# EPICS substitutions: iocs/simple-power-pmac/labApp/Db/lab_expanded.substitutions
# This file was automatically generated on Fri 25 May 2018 08:06:14 BST from
# source: /home/hgv27681/R3.14.12.3/support/pmac/etc/makeIocs/lab.xml
#
# *** Please do not edit this file: edit the source file instead. ***
#

# Macros:
#  PORT      The asyn port for the pmac controller
#  P         PV Prefix
#  NAXES     Number of axes
#  TIMEOUT   Timeout for controller communication
#  FEEDRATE  feedrate below which we go into error
#  CSG0      Name for Coordinate System Group 0
#  CSG1      Name for Coordinate System Group 1
#  CSG2      Name for Coordinate System Group 2
#  CSG3      Name for Coordinate System Group 3
#  CSG4      Name for Coordinate System Group 4
#  CSG5      Name for Coordinate System Group 5
#  CSG6      Name for Coordinate System Group 6
#  CSG7      Name for Coordinate System Group 7
file $(PMAC)/db/pmacController.template
{
pattern { PORT, P, NAXES, TIMEOUT, FEEDRATE, CSG0, CSG1, CSG2, CSG3, CSG4, CSG5, CSG6, CSG7 }
    { "Brick", "BRICK1", "8", "4", "100", "", "", "", "", "", "", "", "" }
}

# Macros:
#  PORT  The asyn port for the pmac controller
#  P     PV Prefix
file $(PMAC)/db/powerPmacStatus.template
{
pattern { PORT, P }
    { "Brick", "BRICK1" }
}

# Macros:
#  PMAC  Pmac/Geobrick name
#  AXIS  Axis number
#  PORT  Asyn port
file $(PMAC)/db/pmacStatusAxis.template
{
pattern { PMAC, AXIS, PORT }
    { "BRICK1", "1", "Brick" }
    { "BRICK1", "2", "Brick" }
    { "BRICK1", "3", "Brick" }
    { "BRICK1", "4", "Brick" }
    { "BRICK1", "5", "Brick" }
    { "BRICK1", "6", "Brick" }
    { "BRICK1", "7", "Brick" }
    { "BRICK1", "8", "Brick" }
}

# Macros:
#  P                Device Prefix
#  M                Device Suffix
#  PORT             Delta tau motor controller
#  ADDR             Address on controller
#  DESC             Description, displayed on EDM screen
#  MRES             Motor Step Size (EGU)
#  VELO             Velocity (EGU/s)
#  PREC             Display Precision
#  EGU              Engineering Units
#  TWV              Tweak Step Size (EGU)
#  DTYP             DTYP of record
#  DIR              User Direction
#  VBAS             Base Velocity (EGU/s)
#  VMAX             Max Velocity (EGU/s), defaults to VELO
#  ACCL             Seconds to Velocity
#  BDST             BL Distance (EGU)
#  BVEL             BL Velocity (EGU/s)
#  BACC             BL Seconds to Veloc.
#  DHLM             Dial High Limit
#  DLLM             Dial Low Limit
#  HLM              User High Limit
#  LLM              User Low Limit
#  HLSV             HW Lim. Violation Svr
#  INIT             Startup commands
#  SREV             Steps per Revolution
#  RRES             Readback Step Size (EGU)
#  ERES             Encoder Step Size (EGU)
#  JAR              Jog Acceleration (EGU/s^2)
#  UEIP             Use Encoder If Present
#  URIP             Use RDBL If Present
#  RDBL             Readback Location, set URIP = 1 if you specify this
#  RLNK             Readback output link
#  RTRY             Max retry count
#  DLY              Readback settle time (s)
#  OFF              User Offset (EGU)
#  RDBD             Retry Deadband (EGU)
#  FOFF             Freeze Offset, 0=variable, 1=frozen
#  ADEL             Alarm monitor deadband (EGU)
#  NTM              New Target Monitor, only set to 0 for soft motors
#  FEHIGH           HIGH limit for following error
#  FEHIHI           HIHI limit for following error
#  FEHHSV           HIHI alarm severity for following error
#  FEHSV            HIGH alarm severity for following error
#  SCALE            Scale factor, if pmacSetAxisScale is used this should be set
#  HOMEVIS          If 1 then home is visible on the gui
#  HOMEVISSTR       If HOMEVIS=0, then display this text on the gui instead
#  name             Object name and gui association name
#  alh              Set this to alh to add the motor to the alarm handler and send emails,
#  gda_name         Name to export this as to GDA
#  gda_desc         Description to export this as to GDA
#  SPORT            Delta tau motor controller comms port
#  HOME             Prefix for autohome instance. Defaults to $(P). If unspecified,
#  ALLOW_HOMED_SET  Set to a blank to allow this axis to have its homed
file $(PMAC)/db/dls_pmac_asyn_motor.template
{
pattern { P, M, PORT, ADDR, DESC, MRES, VELO, PREC, EGU, TWV, DTYP, DIR, VBAS, VMAX, ACCL, BDST, BVEL, BACC, DHLM, DLLM, HLM, LLM, HLSV, INIT, SREV, RRES, ERES, JAR, UEIP, URIP, RDBL, RLNK, RTRY, DLY, OFF, RDBD, FOFF, ADEL, NTM, FEHIGH, FEHIHI, FEHHSV, FEHSV, SCALE, HOMEVIS, HOMEVISSTR, name, alh, gda_name, gda_desc, SPORT, HOME, PMAC, ALLOW_HOMED_SET }
    { "PMAC_BRICK_TEST", ":MOTOR1", "Brick", "1", "Motor 1->A", "1", "20", "3", "mm", "50", "asynMotor", "0", "0", "$(VELO)", "0.5", "0", "0", "", "10000", "-10000", "", "", "MAJOR", "", "1000", "", "", "", "0", "0", "", "", "0", "0", "0", "", "0", "0", "1", "0", "0", "NO_ALARM", "NO_ALARM", "1", "1", "Use motor summary screen", "M1", "None", "", "$(DESC)", "BRICK1port", "$(P)", "BRICK1", "#" }
    { "PMAC_BRICK_TEST", ":MOTOR2", "Brick", "2", "Motor 2->B", "1", "20", "3", "mm", "50", "asynMotor", "0", "0", "$(VELO)", "0.5", "0", "0", "", "10000", "-10000", "", "", "MAJOR", "", "1000", "", "", "", "0", "0", "", "", "0", "0", "0", "", "0", "0", "1", "0", "0", "NO_ALARM", "NO_ALARM", "1", "1", "Use motor summary screen", "M2", "None", "", "$(DESC)", "BRICK1port", "$(P)", "BRICK1", "#" }
    { "PMAC_BRICK_TEST", ":MOTOR3", "Brick", "3", "Motor 3->I JACK 1", "0.001", "20", "3", "mm", "50", "asynMotor", "0", "0", "$(VELO)", "0.5", "0", "0", "", "10000", "-10000", "", "", "MAJOR", "", "1000", "", "", "", "0", "0", "", "", "0", "0", "0", "", "0", "0", "1", "0", "0", "NO_ALARM", "NO_ALARM", "1", "1", "Use motor summary screen", "M3", "None", "", "$(DESC)", "BRICK1port", "$(P)", "BRICK1", "#" }
    { "PMAC_BRICK_TEST", ":MOTOR4", "Brick", "4", "Motor 4->I- JACK 2", "0.001", "20", "3", "mm", "50", "asynMotor", "0", "0", "$(VELO)", "0.5", "0", "0", "", "10000", "-10000", "", "", "MAJOR", "", "1000", "", "", "", "0", "0", "", "", "0", "0", "0", "", "0", "0", "1", "0", "0", "NO_ALARM", "NO_ALARM", "1", "1", "Use motor summary screen", "M4", "None", "", "$(DESC)", "BRICK1port", "$(P)", "BRICK1", "#" }
    { "PMAC_BRICK_TEST", ":MOTOR5", "Brick", "5", "Motor 5", "0.001", "20", "3", "mm", "10", "asynMotor", "0", "0", "$(VELO)", "0.5", "0", "0", "", "10000", "-10000", "", "", "MAJOR", "", "1000", "", "", "", "0", "0", "", "", "0", "0", "0", "", "0", "0", "1", "0", "0", "NO_ALARM", "NO_ALARM", "1", "1", "Use motor summary screen", "M5", "None", "", "$(DESC)", "BRICK1port", "$(P)", "BRICK1", "#" }
    { "PMAC_BRICK_TEST", ":MOTOR6", "Brick", "6", "Motor 6", "0.001", "20", "3", "mm", "10", "asynMotor", "0", "0", "$(VELO)", "0.5", "0", "0", "", "10000", "-10000", "", "", "MAJOR", "", "1000", "", "", "", "0", "0", "", "", "0", "0", "0", "", "0", "0", "1", "0", "0", "NO_ALARM", "NO_ALARM", "1", "1", "Use motor summary screen", "M6", "None", "", "$(DESC)", "BRICK1port", "$(P)", "BRICK1", "#" }
    { "PMAC_BRICK_TEST", ":MOTOR7", "Brick", "7", "Motor 7", "0.001", "20", "3", "mm", "10", "asynMotor", "0", "0", "$(VELO)", "0.5", "0", "0", "", "10000", "-10000", "", "", "MAJOR", "", "1000", "", "", "", "0", "0", "", "", "0", "0", "0", "", "0", "0", "1", "0", "0", "NO_ALARM", "NO_ALARM", "1", "1", "Use motor summary screen", "M7", "None", "", "$(DESC)", "BRICK1port", "$(P)", "BRICK1", "#" }
    { "PMAC_BRICK_TEST", ":MOTOR8", "Brick", "8", "Motor 8", "0.001", "20", "3", "mm", "10", "asynMotor", "0", "0", "$(VELO)", "0.5", "0", "0", "", "10000", "-10000", "", "", "MAJOR", "", "1000", "", "", "", "0", "0", "", "", "0", "0", "0", "", "0", "0", "1", "0", "0", "NO_ALARM", "NO_ALARM", "1", "1", "Use motor summary screen", "M8", "None", "", "$(DESC)", "BRICK1port", "$(P)", "BRICK1", "#" }
}
